Staubli VAL3: Nominal.dtx

public frame fReference = {x=1504.182, y=53.840, z=-415.791, rx=0.201, ry=-0.641, rz=0.004, fatherId=world[0]}
public jointRx jPark = {j1=0.000, j2=0.000, j3=90.000, j4=0.000, j5=90.000, j6=0.000}
public jointRx jJoint = {j1=2.01098, j2=34.80611, j3=88.39690, j4=0.21482, j5=56.14953, j6=-178.11080}
public mdesc mNomSpeed = {accel=100, vel=100, decel=100, tmax=99999, rmax=99999, blend=off, leave=50, reach=50}
public mdesc mSpeed = {tmax=33.3, rmax=100, leave=0.1, reach=0.1, blend=cartesian}
public num nTraj
num nTimeStop
num nTimeStart
num nMode
num nEtat
public pointRx pPoint[13]
  [0] = {x=-35.000, y=0.000, z=0.000, rx=-0.000, ry=0.000, rz=-0.000, shoulder=lefty, elbow=epositive, wrist=wpositive, fatherId=fReference[0]}
  [1] = {x=35.000, y=0.000, z=-1.000, rx=-0.000, ry=0.000, rz=-0.000, shoulder=lefty, elbow=epositive, wrist=wpositive, fatherId=fReference[0]}
  [2] = {x=-34.000, y=0.000, z=-2.000, rx=-0.000, ry=0.000, rz=-0.000, shoulder=lefty, elbow=epositive, wrist=wpositive, fatherId=fReference[0]}
  [3] = {x=34.000, y=0.000, z=-3.000, rx=-0.000, ry=0.000, rz=-0.000, shoulder=lefty, elbow=epositive, wrist=wpositive, fatherId=fReference[0]}
  [4] = {x=-33.000, y=0.000, z=-4.000, rx=-0.000, ry=0.000, rz=-0.000, shoulder=lefty, elbow=epositive, wrist=wpositive, fatherId=fReference[0]}
  [5] = {x=33.000, y=0.000, z=-5.000, rx=-0.000, ry=0.000, rz=-0.000, shoulder=lefty, elbow=epositive, wrist=wpositive, fatherId=fReference[0]}
  [6] = {x=-32.000, y=0.000, z=-6.000, rx=-0.000, ry=0.000, rz=-0.000, shoulder=lefty, elbow=epositive, wrist=wpositive, fatherId=fReference[0]}
  [7] = {x=32.000, y=0.000, z=-7.000, rx=-0.000, ry=0.000, rz=-0.000, shoulder=lefty, elbow=epositive, wrist=wpositive, fatherId=fReference[0]}
  [8] = {x=-31.000, y=0.000, z=-8.000, rx=-0.000, ry=0.000, rz=-0.000, shoulder=lefty, elbow=epositive, wrist=wpositive, fatherId=fReference[0]}
  [9] = {x=31.000, y=0.000, z=-9.000, rx=-0.000, ry=0.000, rz=-0.000, shoulder=lefty, elbow=epositive, wrist=wpositive, fatherId=fReference[0]}
  [10] = {x=-30.000, y=0.000, z=-10.000, rx=-0.000, ry=0.000, rz=-0.000, shoulder=lefty, elbow=epositive, wrist=wpositive, fatherId=fReference[0]}
  [11] = {x=-30.000, y=0.000, z=290.000, rx=-0.000, ry=0.000, rz=-0.000, shoulder=lefty, elbow=epositive, wrist=wpositive, fatherId=fReference[0]}
  [12] = {x=-35.000, y=0.000, z=300.000, rx=-0.000, ry=0.000, rz=-0.000, shoulder=lefty, elbow=epositive, wrist=wpositive, fatherId=fReference[0]}
public tool tTool = {x=-0.047, y=0.112, z=264.182, rx=180.000, ry=0.000, rz=-0.000, fatherId=flange[0], ioLink=valve1}
